(* Logix 5000 project; controller CLP_AB vendor 1 type 14 code 79 rev 17.4; software revision 17.01 *)

TASK DeviceNet (continuous, watchdog 500 ms) : DeviceN
TASK Initialize_speed (event, rate 10 ms, priority 10, watchdog 500 ms) : Initialize_Data
TASK MainTask (periodic, rate 41 ms, priority 10, watchdog 500 ms) : Camera_Trigger

MODULES
   Local : vendor 1 type 14 code 79 (ICP 0, rev 17.4)
      DN : vendor 1 type 12 code 14 (ICP 2, rev 7.3, Output RPI 20 ms, Input RPI 20 ms)
      Ethernet : 1756-ENBT (Ethernet 192.168.0.4, ICP 3, rev 4.1)
         Camera_Sensor : ETHERNET-MODULE (Ethernet 192.168.0.3, rev 1.1, Output RPI 25 ms)   // Banner
      LocalSERCOS : vendor 1 type 16 code 14 (ICP 1, rev 17.2, MotionAsync RPI 25 ms, MotionEvent RPI 1000 ms, MotionSync RPI 2 ms)
         Drive : vendor 1 type 115 code 164 (SERCOS 1, rev 1.1)
END_MODULES

VAR_GLOBAL   (* controller tags *)
   BitTest1 : BOOL;
   BitTest2 : BOOL;
   botao : BOOL;
   dataInitialized : BOOL;
   dir_int : DINT;
   direction : BOOL;
   drive_axis : AXIS_SERVO_DRIVE;
   Emanuel : BOOL;
   encoder : AXIS_SERVO_DRIVE;
   IterationChange : ALIAS FOR Camera_Sensor:I.Data[6].0;
   IterationChanged : BOOL;
   IterationCount : DINT;
   lastIterationCount : DINT;
   MAH_0 : MOTION_INSTRUCTION;
   MAJ_0 : MOTION_INSTRUCTION := (FLAGS := 33554432);
   MAJ_1 : MOTION_INSTRUCTION := (FLAGS := 33554432);
   MAJ_2 : MOTION_INSTRUCTION;
   MAS_0 : MOTION_INSTRUCTION;
   MAS_1 : MOTION_INSTRUCTION := (FLAGS := 33554432);
   MAS_2 : MOTION_INSTRUCTION;
   MGroup : MOTION_GROUP;
   MSF_0 : MOTION_INSTRUCTION;
   MSO_0 : MOTION_INSTRUCTION;
   MSO_1 : MOTION_INSTRUCTION := (FLAGS := -1610612736, EN := 1, DN := 1, STATE := 1);
   OutTest1 : BOOL;
   OutTest2 : BOOL;
   position : ALIAS FOR Camera_Sensor:I.Data[16];
   Ready : ALIAS FOR Camera_Sensor:I.Data[0].4;
   speed : REAL[171];
   speedRate : REAL;
   timer_1 : TIMER := (PRE := 500);
   Trigger_ACK : ALIAS FOR Camera_Sensor:I.Data[0].16;
   trigger_off : TIMER := (PRE := 10);
   trigger_on : TIMER := (PRE := 10);
END_VAR

PROGRAM Camera_Trigger   (* main routine TriggerMain *)
// Trigger
VAR
   Trigger : ALIAS FOR Camera_Sensor:O.Data[0].0;
END_VAR

ROUTINE TriggerMain   (* ladder *)
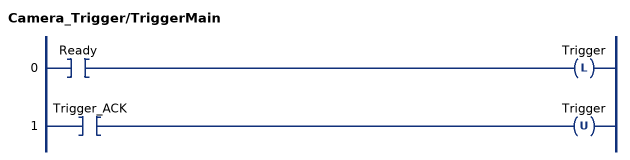
   0: XIC(Ready)OTL(Trigger);
   1: XIC(Trigger_ACK)OTU(Trigger);
END_ROUTINE
END_PROGRAM

PROGRAM Controle   (* main routine malhaAberta *)
VAR
   direcMove : DINT;
   k : DINT;
   timervel : FBD_TIMER;
END_VAR

ROUTINE ControleMain   (* structured text *)
   COP(Camera_Sensor:I.Data[6],IterationCount,32);
   if IterationCount > lastIterationCount then
   	/*Aqui vai o nosso controlador*/
   	if position > 205.0 then
   		speedRate:=.2;
   		direcMove:=1;
   	elsif position < 195.0 then
   		speedRate:=.2;
   		direcMove:=0;
   	else
   		speedRate:=0;
   		MAS(drive_axis,MAS_1,0,0,100,1,0,100,1);
   	end_if;
   	MAJ(drive_axis,MAJ_1,direcMove,speedRate,0,50.0,1,50.0,1,0,50.0,50.0,1,0,0);
   	COP(Camera_Sensor:I.Data[6],lastIterationCount,32);
   end_if;
END_ROUTINE

ROUTINE malhaAberta   (* structured text *)
   // k is the index of the speed vector
   if dataInitialized AND k < 170 then
   	MAJ(drive_axis,MAJ_1,0,speed[k],0,50.0,1,50.0,1,0,50.0,50.0,1,0,0);
   	k:=k + 1;
   end_if;
   
   if k >= 170 then
   	MAS(drive_axis,MAS_1,0,0,100,1,0,100,1);
   	if MAS_1.DN then
   		MSF(drive_axis,MSF_0);
   	end_if;
   end_if;
END_ROUTINE

ROUTINE VeloMain   (* structured text *)
   COP(Camera_Sensor:I.Data[6],IterationCount,32);
   /*MAJ(drive_axis,MAJ_1,0,0.5,0,50.0,1,50.0,1,0,50.0,50.0,1,0,0);
   timervel.TimerEnable:=1;
   TONR(timervel);
   MAS(drive_axis,MAS_1,All,0,100,1,0,100,1);
   MSF(drive_axis,MSF_0);
   */
   	//MSO(drive_axis,MSO_1);
   	timervel.PRE:=20000;
   	if (MSO_1.EN AND timervel.ACC < 20000) then
   		if (NOT timervel.DN) then
   			timervel.TimerEnable:=1;
   			MAJ(drive_axis,MAJ_1,0,0.2,0,50.0,1,50.0,1,0,50.0,50.0,1,0,0);
   			TONR(timervel);
   		end_if;
   	end_if;
   	if (timervel.DN) then
   		MAS(drive_axis,MAS_1,All,0,100,1,0,100,1);
   	end_if;
   	if (MAS_1.EN) then
   		MSF(drive_axis,MSF_0);
   	end_if;
   
END_ROUTINE
END_PROGRAM

PROGRAM Controle1   (* main routine VeloMain *)
VAR
   direcMove : DINT;
   timervel : FBD_TIMER;
END_VAR

ROUTINE ControleMain   (* structured text *)
   COP(Camera_Sensor:I.Data[6],IterationCount,32);
   if IterationCount > lastIterationCount then
   	/*Aqui vai o nosso controlador*/
   	if position > 205.0 then
   		speedRate:=.2;
   		direcMove:=1;
   	elsif position < 195.0 then
   		speedRate:=.2;
   		direcMove:=0;
   	else
   		speedRate:=0;
   		MAS(drive_axis,MAS_1,0,0,100,1,0,100,1);
   	end_if;
   	MAJ(drive_axis,MAJ_1,direcMove,speedRate,0,50.0,1,50.0,1,0,50.0,50.0,1,0,0);
   	COP(Camera_Sensor:I.Data[6],lastIterationCount,32);
   end_if;
END_ROUTINE

ROUTINE VeloMain   (* structured text *)
   COP(Camera_Sensor:I.Data[6],IterationCount,32);
   /*MAJ(drive_axis,MAJ_1,0,0.5,0,50.0,1,50.0,1,0,50.0,50.0,1,0,0);
   timervel.TimerEnable:=1;
   TONR(timervel);
   MAS(drive_axis,MAS_1,All,0,100,1,0,100,1);
   MSF(drive_axis,MSF_0);
   */
   	//MSO(drive_axis,MSO_1);
   	timervel.PRE:=20000;
   	if (MSO_1.EN AND timervel.ACC < 20000) then
   		if (NOT timervel.DN) then
   			timervel.TimerEnable:=1;
   			MAJ(drive_axis,MAJ_1,0,0.2,0,50.0,1,50.0,1,0,50.0,50.0,1,0,0);
   			TONR(timervel);
   		end_if;
   	end_if;
   	if (timervel.DN) then
   		MAS(drive_axis,MAS_1,All,0,100,1,0,100,1);
   	end_if;
   	if (MAS_1.EN) then
   		MSF(drive_axis,MSF_0);
   	end_if;
   
END_ROUTINE
END_PROGRAM

PROGRAM DeviceN   (* main routine InitDNetST *)

ROUTINE InitDNetST   (* structured text *)
   Local:2:O.CommandRegister.Run [:=] 1;
   if NOT dataInitialized then
   	EVENT(Initialize_speed);
   end_if;
   
END_ROUTINE
END_PROGRAM

PROGRAM Initialize_Data   (* main routine Init *)

ROUTINE Init   (* structured text *)
   /* Universidade de Brasilia
   Trabalho de Graduacao em Engenharia Mecatronica
   Alunos:
   Ataias Pereira Reis 10/0093817
   Emanuel Pereira Barroso Neto 11/0115716
   This code must be executed only once. */
   
   MSO(drive_axis,MSO_1);
   
   speed[0] := 0.0;
   speed[1] := 0.0;
   speed[2] := 0.0;
   speed[3] := 0.0;
   speed[4] := 0.0;
   speed[5] := 0.0;
   speed[6] := 0.0;
   speed[7] := 0.0;
   speed[8] := 0.0;
   speed[9] := 0.0;
   speed[10] := 0.0;
   speed[11] := 0.0;
   speed[12] := 0.0;
   speed[13] := 0.0;
   speed[14] := 0.0;
   speed[15] := 0.0;
   speed[16] := 0.0;
   speed[17] := 0.0;
   speed[18] := 0.0;
   speed[19] := 0.0;
   speed[20] := 0.0;
   speed[21] := 0.0147026554205;
   speed[22] := 0.0547055820855;
   speed[23] := 0.114361720023;
   speed[24] := 0.18111091036;
   speed[25] := 0.251809893147;
   speed[26] := 0.32607467121;
   speed[27] := 0.403453064793;
   speed[28] := 0.483471620607;
   speed[29] := 0.565658044965;
   speed[30] := 0.649536805548;
   speed[31] := 0.734630464537;
   speed[32] := 0.820458741642;
   speed[33] := 0.906543473223;
   speed[34] := 0.992424061587;
   speed[35] := 1.07765619092;
   speed[36] := 1.16189824235;
   speed[37] := 1.24456943015;
   speed[38] := 1.32036725857;
   speed[39] := 1.3812552175;
   speed[40] := 1.43231065067;
   speed[41] := 1.48663214948;
   speed[42] := 1.54839415747;
   speed[43] := 1.61599008767;
   speed[44] := 1.68757723373;
   speed[45] := 1.7613579514;
   speed[46] := 1.83569169336;
   speed[47] := 1.90907847349;
   speed[48] := 1.9801747816;
   speed[49] := 2.04784594244;
   speed[50] := 2.11113619377;
   speed[51] := 2.16944638193;
   speed[52] := 2.22182598313;
   speed[53] := 2.26825099412;
   speed[54] := 2.30985215012;
   speed[55] := 2.34320587986;
   speed[56] := 2.36620871737;
   speed[57] := 2.38071882377;
   speed[58] := 2.38672834648;
   speed[59] := 2.38430263817;
   speed[60] := 2.37407699776;
   speed[61] := 2.35619724752;
   speed[62] := 2.33055863496;
   speed[63] := 2.29754175796;
   speed[64] := 2.25797832185;
   speed[65] := 2.21262636405;
   speed[66] := 2.16123527696;
   speed[67] := 2.10467481035;
   speed[68] := 2.04388225087;
   speed[69] := 1.97863997419;
   speed[70] := 1.90950133568;
   speed[71] := 1.83693203375;
   speed[72] := 1.7619821587;
   speed[73] := 1.686412295;
   speed[74] := 1.60932227957;
   speed[75] := 1.53031257908;
   speed[76] := 1.45140199977;
   speed[77] := 1.37297157979;
   speed[78] := 1.29394180319;
   speed[79] := 1.2157528212;
   speed[80] := 1.1408355106;
   speed[81] := 1.06779007087;
   speed[82] := 0.995420551475;
   speed[83] := 0.924581999131;
   speed[84] := 0.855323010933;
   speed[85] := 0.788477897412;
   speed[86] := 0.726538190521;
   speed[87] := 0.66801109369;
   speed[88] := 0.607741032753;
   speed[89] := 0.547567758592;
   speed[90] := 0.493301637758;
   speed[91] := 0.440419162243;
   speed[92] := 0.387507265216;
   speed[93] := 0.338400915621;
   speed[94] := 0.291658541896;
   speed[95] := 0.248512542153;
   speed[96] := 0.209796973955;
   speed[97] := 0.172530018125;
   speed[98] := 0.141664432169;
   speed[99] := 0.11599366767;
   speed[100] := 0.087107967923;
   speed[101] := 0.0627295944751;
   speed[102] := 0.0490272896769;
   speed[103] := 0.0374349286012;
   speed[104] := 0.0234408281723;
   speed[105] := 0.0103613796074;
   speed[106] := 0.0;
   speed[107] := 0.0;
   speed[108] := 0.0;
   speed[109] := 0.0;
   speed[110] := 0.0;
   speed[111] := 0.0;
   speed[112] := 0.0;
   speed[113] := 0.0;
   speed[114] := 0.0;
   speed[115] := 0.0;
   speed[116] := 0.0;
   speed[117] := 0.0;
   speed[118] := 0.0;
   speed[119] := 0.0;
   speed[120] := 0.0;
   speed[121] := 0.0;
   speed[122] := 0.0;
   speed[123] := 0.0;
   speed[124] := 0.0;
   speed[125] := 0.0;
   speed[126] := 0.0;
   speed[127] := 0.0;
   speed[128] := 0.0;
   speed[129] := 0.0;
   speed[130] := 0.0;
   speed[131] := 0.0;
   speed[132] := 0.0;
   speed[133] := 0.0;
   speed[134] := 0.0;
   speed[135] := 0.0;
   speed[136] := 0.0;
   speed[137] := 0.0;
   speed[138] := 0.0;
   speed[139] := 0.0;
   speed[140] := 0.0;
   speed[141] := 0.0;
   speed[142] := 0.0;
   speed[143] := 0.0;
   speed[144] := 0.0;
   speed[145] := 0.0;
   speed[146] := 0.0;
   speed[147] := 0.0;
   speed[148] := 0.0;
   speed[149] := 0.0;
   speed[150] := 0.0;
   speed[151] := 0.0;
   speed[152] := 0.0;
   speed[153] := 0.0;
   speed[154] := 0.0;
   speed[155] := 0.0;
   speed[156] := 0.0;
   speed[157] := 0.0;
   speed[158] := 0.0;
   speed[159] := 0.0;
   speed[160] := 0.0;
   speed[161] := 0.0;
   speed[162] := 0.0;
   speed[163] := 0.0;
   speed[164] := 0.0;
   speed[165] := 0.0;
   speed[166] := 0.0;
   speed[167] := 0.0;
   speed[168] := 0.0;
   speed[169] := 0.0;
   speed[170] := 0.0;
   
   dataInitialized := 1; //true
END_ROUTINE
END_PROGRAM

PROGRAM MainProgram   (* main routine MainRoutineST *)

ROUTINE MainRoutine   (* ladder *)
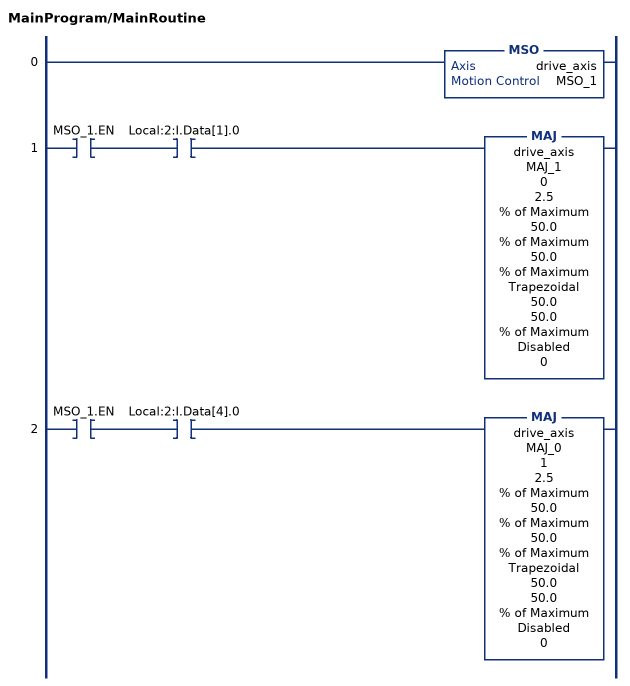
   0: MSO(drive_axis,MSO_1);
   1: XIC(MSO_1.EN)XIC(Local:2:I.Data[1].0)MAJ(drive_axis,MAJ_1,0,2.5,% of Maximum,50.0,% of Maximum,50.0,% of Maximum,Trapezoidal,50.0,50.0,% of Maximum,Disabled,0);
   2: XIC(MSO_1.EN)XIC(Local:2:I.Data[4].0)MAJ(drive_axis,MAJ_0,1,2.5,% of Maximum,50.0,% of Maximum,50.0,% of Maximum,Trapezoidal,50.0,50.0,% of Maximum,Disabled,0);
END_ROUTINE

ROUTINE MainRoutineST   (* structured text *)
   MSO(drive_axis,MSO_1);
   IF MSO_1.EN AND Local:2:I.Data[1].0 THEN
   	MAJ(drive_axis,MAJ_1,0,2.5,1,50.0,1,50.0,1,0,50.0,50.0,1,0,0);
   END_IF;
   IF MSO_1.EN AND Local:2:I.Data[4].0 THEN
   	MAJ(drive_axis,MAJ_0,1,2.5,1,50.0,1,50.0,1,0,50.0,50.0,1,0,0);
   END_IF;
END_ROUTINE
END_PROGRAM

PROGRAM Parada   (* main routine parada *)

ROUTINE parada   (* ladder *)
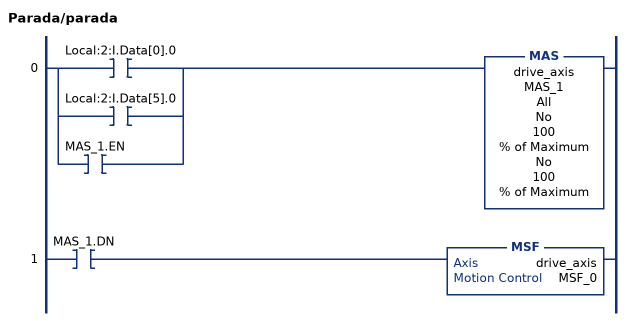
   0: [XIC(Local:2:I.Data[0].0) ,[XIC(Local:2:I.Data[5].0) ,XIC(MAS_1.EN) ] ]MAS(drive_axis,MAS_1,All,No,100,% of Maximum,No,100,% of Maximum);
   1: XIC(MAS_1.DN)MSF(drive_axis,MSF_0);
END_ROUTINE
END_PROGRAM
